PROGRAM Stn1
VAR

	start1: BOOL;
	reset1: BOOL;

	Stn1ProcessFE: F_TRIG;
	Stn1ProcessRE: R_TRIG;
	bCutStn1ProcessHalt: BOOL;
	DoorClose1: R_TRIG;
	bStn1DoorClamp: BOOL;

END_VAR
VAR // added by the converter: edge detectors and wires of the graphical bodies
    _w1, _w2 : ANY;
END_VAR

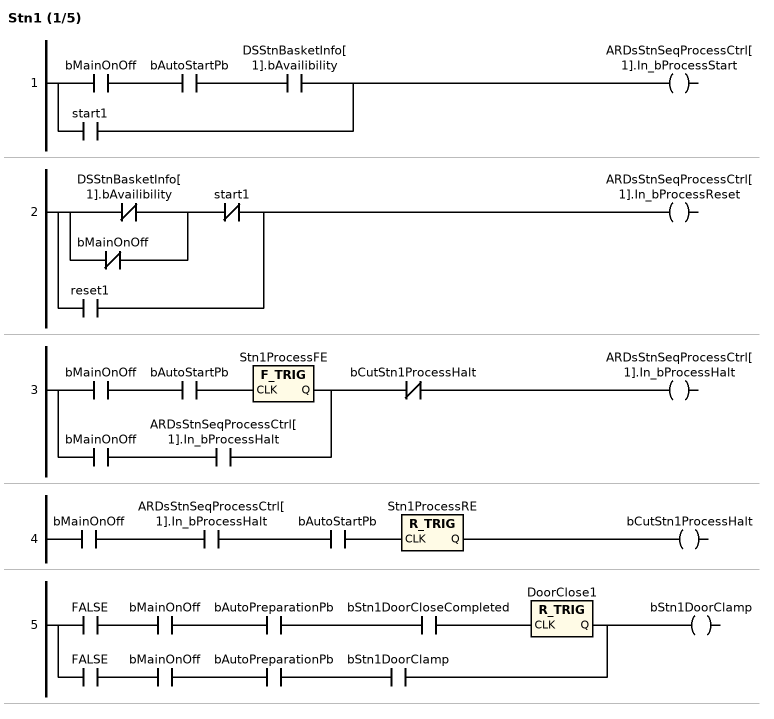
// NETWORK 1
ARDsStnSeqProcessCtrl[1].In_bProcessStart := bMainOnOff AND bAutoStartPb AND DSStnBasketInfo[1].bAvailibility OR start1;

// NETWORK 2
ARDsStnSeqProcessCtrl[1].In_bProcessReset := (NOT DSStnBasketInfo[1].bAvailibility OR NOT bMainOnOff) AND NOT start1 OR reset1;

// NETWORK 3
Stn1ProcessFE(CLK := bMainOnOff AND bAutoStartPb); // F_TRIG
ARDsStnSeqProcessCtrl[1].In_bProcessHalt := (Stn1ProcessFE.Q OR bMainOnOff AND ARDsStnSeqProcessCtrl[1].In_bProcessHalt) AND NOT bCutStn1ProcessHalt;

// NETWORK 4
Stn1ProcessRE(CLK := bMainOnOff AND ARDsStnSeqProcessCtrl[1].In_bProcessHalt AND bAutoStartPb); // R_TRIG
bCutStn1ProcessHalt := Stn1ProcessRE.Q;

// NETWORK 5
DoorClose1(CLK := (FALSE AND bMainOnOff AND bAutoPreparationPb) AND bStn1DoorCloseCompleted); // R_TRIG
bStn1DoorClamp := DoorClose1.Q OR (FALSE AND bMainOnOff AND bAutoPreparationPb) AND bStn1DoorClamp;

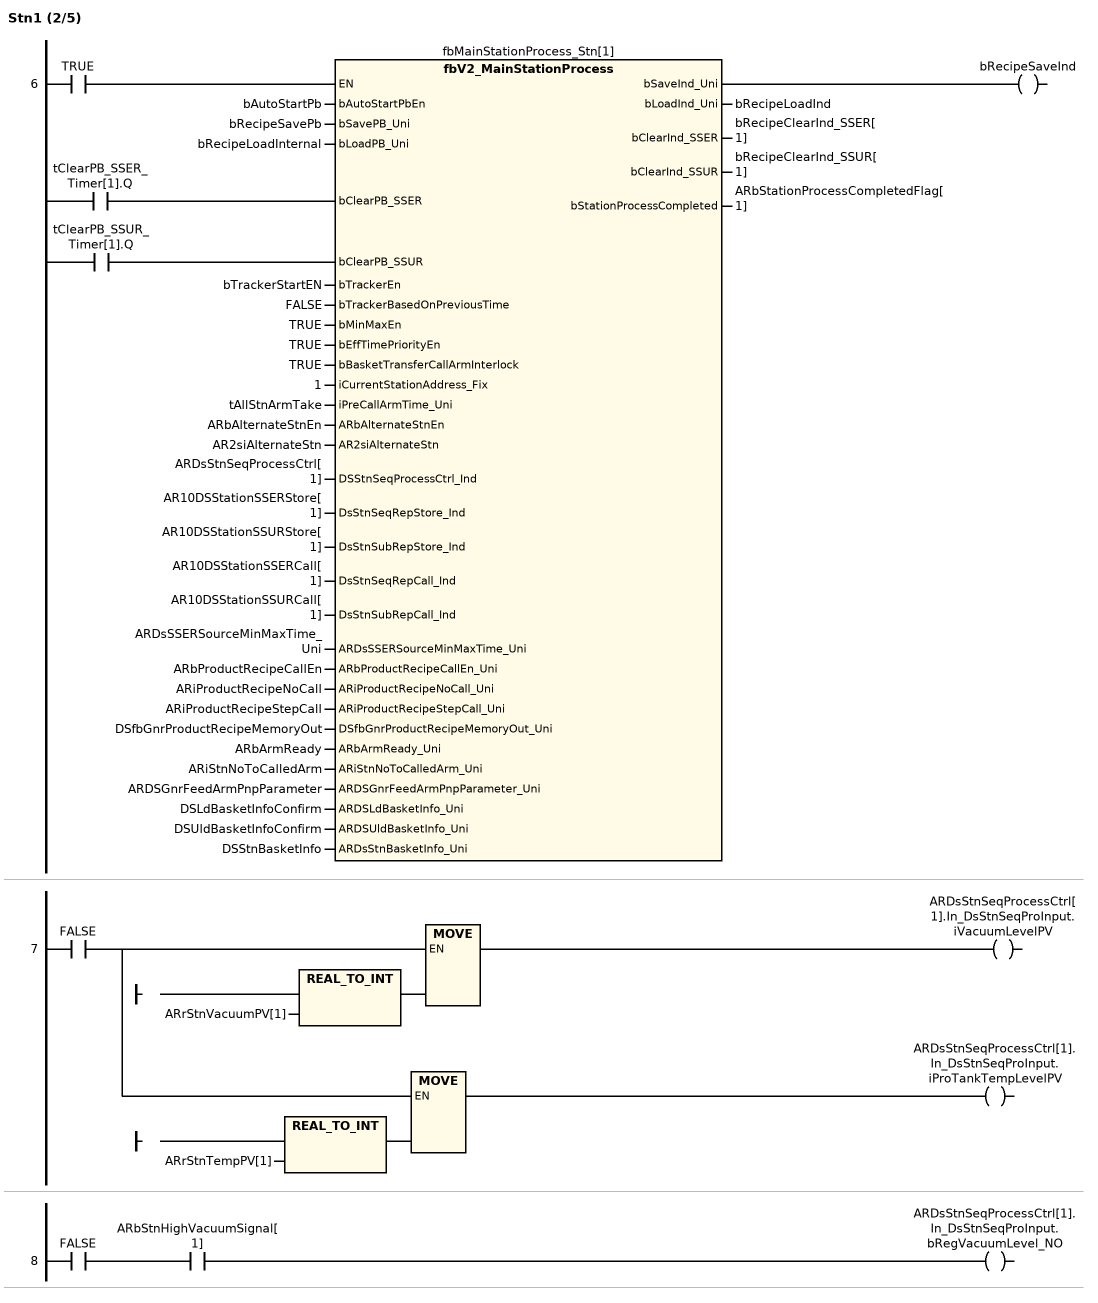
// NETWORK 6
fbMainStationProcess_Stn[1](
    bAutoStartPbEn := bAutoStartPb,
    bSavePB_Uni := bRecipeSavePb,
    bLoadPB_Uni := bRecipeLoadInternal,
    bClearPB_SSER := tClearPB_SSER_Timer[1].Q,
    bClearPB_SSUR := tClearPB_SSUR_Timer[1].Q,
    bTrackerEn := bTrackerStartEN,
    bTrackerBasedOnPreviousTime := FALSE,
    bMinMaxEn := TRUE,
    bEffTimePriorityEn := TRUE,
    bBasketTransferCallArmInterlock := TRUE,
    iCurrentStationAddress_Fix := 1,
    iPreCallArmTime_Uni := tAllStnArmTake,
    ARbAlternateStnEn := ARbAlternateStnEn,
    AR2siAlternateStn := AR2siAlternateStn,
    DSStnSeqProcessCtrl_Ind := ARDsStnSeqProcessCtrl[1],
    DsStnSeqRepStore_Ind := AR10DSStationSSERStore[1],
    DsStnSubRepStore_Ind := AR10DSStationSSURStore[1],
    DsStnSeqRepCall_Ind := AR10DSStationSSERCall[1],
    DsStnSubRepCall_Ind := AR10DSStationSSURCall[1],
    ARDsSSERSourceMinMaxTime_Uni := ARDsSSERSourceMinMaxTime_Uni,
    ARbProductRecipeCallEn_Uni := ARbProductRecipeCallEn,
    ARiProductRecipeNoCall_Uni := ARiProductRecipeNoCall,
    ARiProductRecipeStepCall_Uni := ARiProductRecipeStepCall,
    DSfbGnrProductRecipeMemoryOut_Uni := DSfbGnrProductRecipeMemoryOut,
    ARbArmReady_Uni := ARbArmReady,
    ARiStnNoToCalledArm_Uni := ARiStnNoToCalledArm,
    ARDSGnrFeedArmPnpParameter_Uni := ARDSGnrFeedArmPnpParameter,
    ARDSLdBasketInfo_Uni := DSLdBasketInfoConfirm,
    ARDSUldBasketInfo_Uni := DSUldBasketInfoConfirm,
    ARDsStnBasketInfo_Uni := DSStnBasketInfo,
    bLoadInd_Uni => bRecipeLoadInd,
    bClearInd_SSER => bRecipeClearInd_SSER[1],
    bClearInd_SSUR => bRecipeClearInd_SSUR[1],
    bStationProcessCompleted => ARbStationProcessCompletedFlag[1]); // fbV2_MainStationProcess
bRecipeSaveInd := fbMainStationProcess_Stn[1].bSaveInd_Uni;

// NETWORK 7
IF FALSE THEN _w1 := REAL_TO_INT(ARrStnVacuumPV[1]); END_IF
ARDsStnSeqProcessCtrl[1].In_DsStnSeqProInput.iVacuumLevelPV := _w1;
IF FALSE THEN _w2 := REAL_TO_INT(ARrStnTempPV[1]); END_IF
ARDsStnSeqProcessCtrl[1].In_DsStnSeqProInput.iProTankTempLevelPV := _w2;

// NETWORK 8
ARDsStnSeqProcessCtrl[1].In_DsStnSeqProInput.bRegVacuumLevel_NO := FALSE AND ARbStnHighVacuumSignal[1];

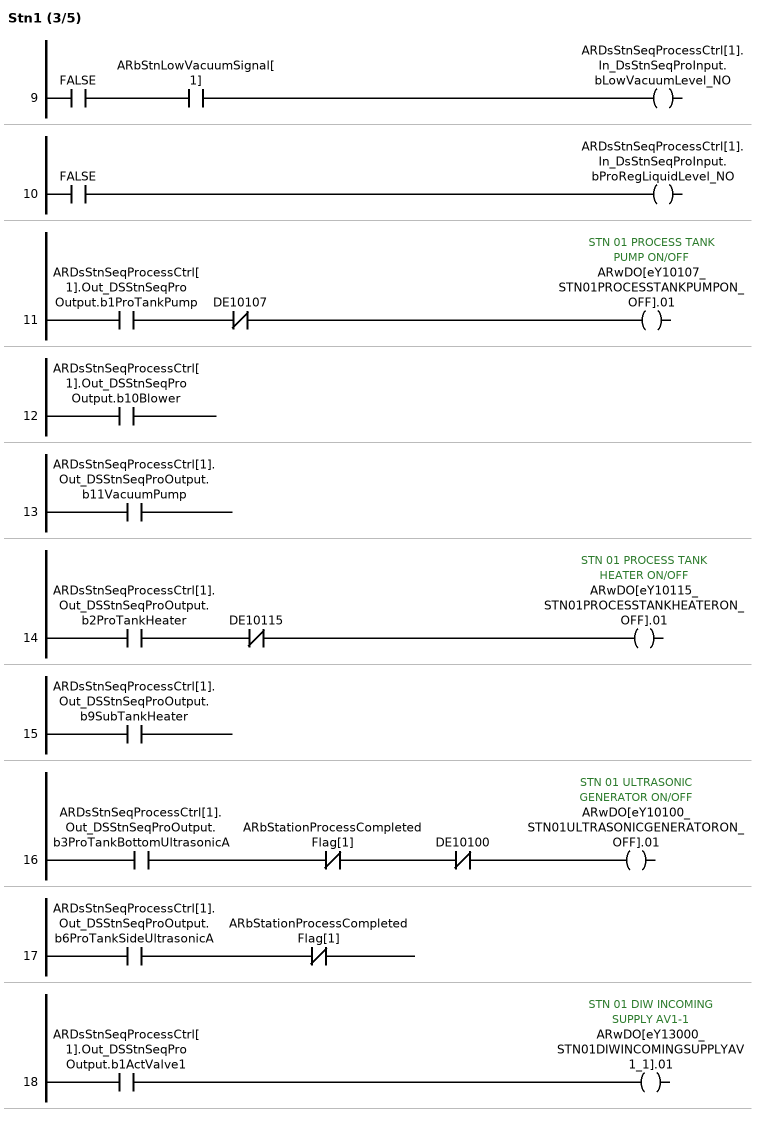
// NETWORK 9
ARDsStnSeqProcessCtrl[1].In_DsStnSeqProInput.bLowVacuumLevel_NO := FALSE AND ARbStnLowVacuumSignal[1];

// NETWORK 10
ARDsStnSeqProcessCtrl[1].In_DsStnSeqProInput.bProRegLiquidLevel_NO := FALSE;

// NETWORK 11
//   ARwDO[eY10107_STN01PROCESSTANKPUMPON_OFF].01: STN 01 PROCESS TANK PUMP ON/OFF
ARwDO[eY10107_STN01PROCESSTANKPUMPON_OFF].01 := ARDsStnSeqProcessCtrl[1].Out_DSStnSeqProOutput.b1ProTankPump AND NOT DE10107;

// NETWORK 12
(* ARDsStnSeqProcessCtrl[1].Out_DSStnSeqProOutput.b10Blower; not connected *)

// NETWORK 13
(* ARDsStnSeqProcessCtrl[1].Out_DSStnSeqProOutput.b11VacuumPump; not connected *)

// NETWORK 14
//   ARwDO[eY10115_STN01PROCESSTANKHEATERON_OFF].01: STN 01 PROCESS TANK HEATER ON/OFF
ARwDO[eY10115_STN01PROCESSTANKHEATERON_OFF].01 := ARDsStnSeqProcessCtrl[1].Out_DSStnSeqProOutput.b2ProTankHeater AND NOT DE10115;

// NETWORK 15
(* ARDsStnSeqProcessCtrl[1].Out_DSStnSeqProOutput.b9SubTankHeater; not connected *)

// NETWORK 16
//   ARwDO[eY10100_STN01ULTRASONICGENERATORON_OFF].01: STN 01 ULTRASONIC GENERATOR ON/OFF
ARwDO[eY10100_STN01ULTRASONICGENERATORON_OFF].01 := ARDsStnSeqProcessCtrl[1].Out_DSStnSeqProOutput.b3ProTankBottomUltrasonicA AND NOT ARbStationProcessCompletedFlag[1] AND NOT DE10100;

// NETWORK 17
(* ARDsStnSeqProcessCtrl[1].Out_DSStnSeqProOutput.b6ProTankSideUltrasonicA AND NOT ARbStationProcessCompletedFlag[1]; result not used *)

// NETWORK 18
//   ARwDO[eY13000_STN01DIWINCOMINGSUPPLYAV1_1].01: STN 01 DIW INCOMING SUPPLY AV1-1
ARwDO[eY13000_STN01DIWINCOMINGSUPPLYAV1_1].01 := ARDsStnSeqProcessCtrl[1].Out_DSStnSeqProOutput.b1ActValve1;

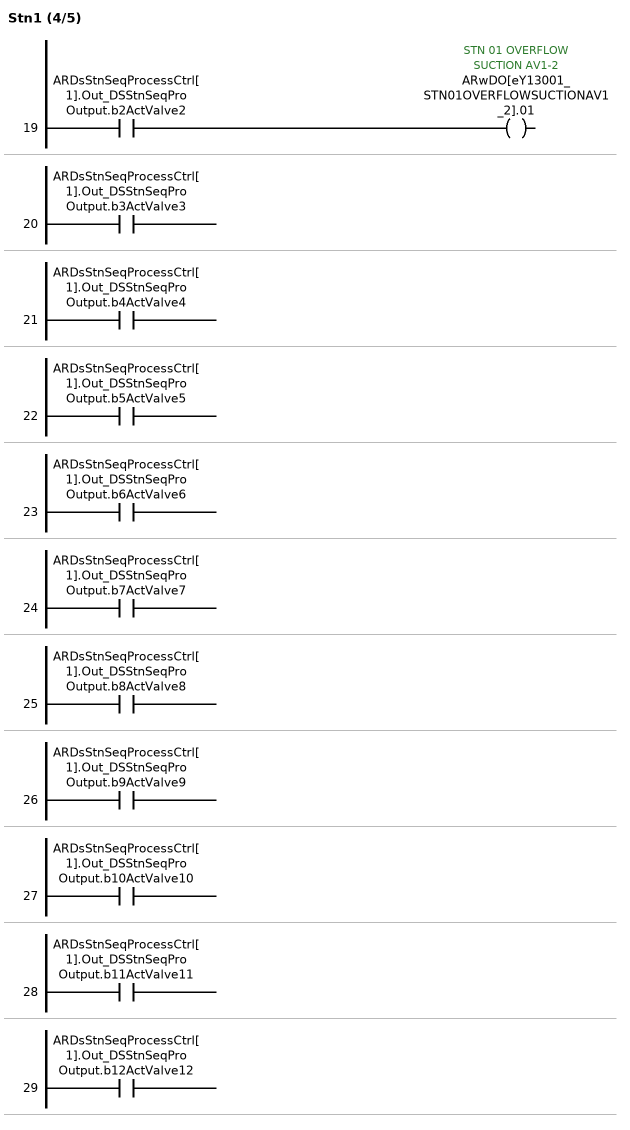
// NETWORK 19
//   ARwDO[eY13001_STN01OVERFLOWSUCTIONAV1_2].01: STN 01 OVERFLOW SUCTION AV1-2
ARwDO[eY13001_STN01OVERFLOWSUCTIONAV1_2].01 := ARDsStnSeqProcessCtrl[1].Out_DSStnSeqProOutput.b2ActValve2;

// NETWORK 20
(* ARDsStnSeqProcessCtrl[1].Out_DSStnSeqProOutput.b3ActValve3; not connected *)

// NETWORK 21
(* ARDsStnSeqProcessCtrl[1].Out_DSStnSeqProOutput.b4ActValve4; not connected *)

// NETWORK 22
(* ARDsStnSeqProcessCtrl[1].Out_DSStnSeqProOutput.b5ActValve5; not connected *)

// NETWORK 23
(* ARDsStnSeqProcessCtrl[1].Out_DSStnSeqProOutput.b6ActValve6; not connected *)

// NETWORK 24
(* ARDsStnSeqProcessCtrl[1].Out_DSStnSeqProOutput.b7ActValve7; not connected *)

// NETWORK 25
(* ARDsStnSeqProcessCtrl[1].Out_DSStnSeqProOutput.b8ActValve8; not connected *)

// NETWORK 26
(* ARDsStnSeqProcessCtrl[1].Out_DSStnSeqProOutput.b9ActValve9; not connected *)

// NETWORK 27
(* ARDsStnSeqProcessCtrl[1].Out_DSStnSeqProOutput.b10ActValve10; not connected *)

// NETWORK 28
(* ARDsStnSeqProcessCtrl[1].Out_DSStnSeqProOutput.b11ActValve11; not connected *)

// NETWORK 29
(* ARDsStnSeqProcessCtrl[1].Out_DSStnSeqProOutput.b12ActValve12; not connected *)

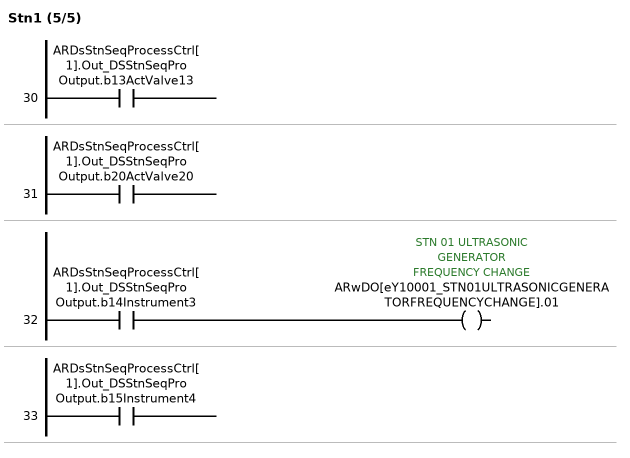
// NETWORK 30
(* ARDsStnSeqProcessCtrl[1].Out_DSStnSeqProOutput.b13ActValve13; not connected *)

// NETWORK 31
(* ARDsStnSeqProcessCtrl[1].Out_DSStnSeqProOutput.b20ActValve20; not connected *)

// NETWORK 32
//   ARwDO[eY10001_STN01ULTRASONICGENERATORFREQUENCYCHANGE].01: STN 01 ULTRASONIC GENERATOR FREQUENCY CHANGE
ARwDO[eY10001_STN01ULTRASONICGENERATORFREQUENCYCHANGE].01 := ARDsStnSeqProcessCtrl[1].Out_DSStnSeqProOutput.b14Instrument3;

// NETWORK 33
(* ARDsStnSeqProcessCtrl[1].Out_DSStnSeqProOutput.b15Instrument4; not connected *)

END_PROGRAM

(* stored: Version 1.1.0.1, ProductVersion 3.1.4024.12
   POU Stn1: Id {f6a77222-d84e-4ba1-bb59-48c248f7649a}, SpecialFunc None *)
